FUNCTION RadToDeg : LREAL
VAR_INPUT
    radians : LREAL;
END_VAR
VAR
END_VAR

RadToDeg := radians / PI * 180.0;

END_FUNCTION

(* stored: Version 1.1.0.1, ProductVersion 3.1.4018.2
   POU RadToDeg: Id {dba2fc67-fc85-404b-acf9-714d94ed067b}, SpecialFunc None *)
